// TIA Portal V15 export
// export: Created 2018-06-08T08:02:20.3305421Z, ExportSetting WithDefaults, WithReadOnly, DisplayName Totally Integrated Automation Portal, DisplayVersion V15, DisplayName TIA Portal Openness, DisplayVersion V15, DisplayName STEP 7 Professional, DisplayVersion V15, DisplayName WinCC Professional, DisplayVersion V15
ORGANIZATION_BLOCK "Main"   // OB1, STL, ProgramCycle
TITLE = "Main Program Sweep (Cycle)"
{ S7_Optimized_Access := 'FALSE' }
VERSION : 0.1
// stored: AutoNumber false, CodeModifiedDate 2018-06-08T08:01:58.298282Z, CompileDate 2018-06-08T08:01:58.2972819Z, CreationDate 2018-05-29T13:31:39.8908501Z, InterfaceModifiedDate 2007-08-03T16:55:08.419547Z, IsConsistent true, IsKnowHowProtected false, IsWriteProtected false, ModifiedDate 2018-06-08T08:01:58.298282Z, ParameterModified 2007-08-03T16:55:08.419547Z, StructureModified 2007-08-03T16:55:08.419547Z
   VAR_TEMP
      OB1_EV_CLASS : Byte;   // Bits 0-3 = 1 (Coming event), Bits 4-7 = 1 (Event class 1)
      OB1_SCAN_1 : Byte;   // 1 (Cold restart scan 1 of OB 1), 3 (Scan 2-n of OB 1)
      OB1_PRIORITY : Byte;   // Priority of OB Execution
      OB1_OB_NUMBR : Byte;   // 1 (Organization block 1, OB1)
      OB1_RESERVED_1 : Byte;   // Reserved for system
      OB1_RESERVED_2 : Byte;   // Reserved for system
      OB1_PREV_CYCLE : Int;   // Cycle time of previous OB1 scan (milliseconds)
      OB1_MIN_CYCLE : Int;   // Minimum cycle time of OB1 (milliseconds)
      OB1_MAX_CYCLE : Int;   // Maximum cycle time of OB1 (milliseconds)
      OB1_DATE_TIME : Date_And_Time;   // Date and time OB1 started
   END_VAR
BEGIN

NETWORK
TITLE = Main
// comment
	CALL	Main_Program
END_ORGANIZATION_BLOCK
